		hr := F_VN_ResizeImage(ipImageIn,
							   ipImageForVideoRingBuffer,
							   ImageSmallWidth,
							   ImageSmallHeight,
							   1,
							   hr);
	ELSE
		hr := F_VN_CopyImage(ipImageIn, ipImageForVideoRingBuffer, hr);
	END_IF

	// Check to see if images are in memory
	//hr := FW_SafeRelease(ADR(BufferImageRing[BufferIndex]));
	//IF BufferImageRing[BufferIndex] <> 0 THEN
	//	FW_SafeRelease(ADR(BufferImageRing[BufferIndex]));
	//END_IF
	
	
	hrWD1		:= F_VN_StartRelWatchdog(tStop1, S_OK);
	hr			:= F_VN_CopyImage(ipImageForVideoRingBuffer, BufferImageRing[BufferIndex], S_OK);
	hrWD1		:= F_VN_StopWatchdog(hrWD1, tRest => tRest1);
	BufferIndex := BufferIndex + 1;
	IF BufferIndex > Parameters_Vision.MAX_NUMBER_IMAGES_2_VIDEO THEN
		BufferIndex := 1;
	END_IF
END_IF
END_METHOD

PROPERTY AlarmDelayTime : TIME
SET
_AlarmDelayTime := AlarmDelayTime;
END_SET
END_PROPERTY

PROPERTY CameraID : UINT
SET
_CameraID := CameraID;
END_SET
END_PROPERTY

PROPERTY FramesPerSecond : UINT
SET
_FramesPerSecond := FramesPerSecond;
END_SET
END_PROPERTY

PROPERTY ImageReductionFactor : LREAL
SET
_ImageReductionFactor := ImageReductionFactor;
END_SET
END_PROPERTY

PROPERTY ImageSourceDirectory : STRING
SET
_ImageSourceDirectory := ImageSourceDirectory;
END_SET
END_PROPERTY

PROPERTY VideoOutputDirectory : STRING
SET
_VideoOutputDirectory := VideoOutputDirectory;
END_SET
END_PROPERTY

METHOD WriteImage : BOOL
VAR_INPUT
	BufferImageSaveNameIndex : INT;
	Index					 : INT;
END_VAR

VAR
	SysTimeAtImageSave : ULINT;
END_VAR
CASE WriteFileState OF
	0:
		sImageToSaveName := CONCAT(STR1 := _ImageSourceDirectory, '\Image');
		CASE Index OF // Add leading zeros to index number of image name
			0..9:
				sImageToSaveName := CONCAT(sImageToSaveName, '000');
				sImageToSaveName := CONCAT(sImageToSaveName, ULINT_TO_STRING(Index));

			10..99:
				sImageToSaveName := CONCAT(sImageToSaveName, '00');
				sImageToSaveName := CONCAT(sImageToSaveName, ULINT_TO_STRING(Index));

			100..999:
				sImageToSaveName := CONCAT(sImageToSaveName, '0');
				sImageToSaveName := CONCAT(sImageToSaveName, ULINT_TO_STRING(Index));

		ELSE
			sImageToSaveName := CONCAT(sImageToSaveName, ULINT_TO_STRING(Index));
		END_CASE;

		sImageToSaveName	:= CONCAT(sImageToSaveName, '.png');
		ipImageToSave		:= BufferImageRing[BufferImageSaveNameIndex];
		SysTimeAtImageSave	:= F_GetSystemTime();
		WriteFileState		:= 10;

	10:
		// sFilePath must contain the full path, image name and type
		fbWriteImage(ipImage := ipImageToSave, sFilePath := sImageToSaveName, nTimeout := T#500MS,bWrite := TRUE);
		IF NOT fbWriteImage.bBusy THEN
			fbWriteImage(sFilePath := sImageToSaveName, bWrite := FALSE);
			WriteFileState := 0;
			WriteImage := TRUE;
		END_IF

ELSE
	WriteFileState := 0;
END_CASE

(*//bSaveImageNow := FALSE;
WriteImageWaitResult := TRUE;

// sFilePath must contain the full path, image name and type
fbWriteImage(ipImage   := ipImageToSave,
			 sFilePath := sImageToSaveName,
			 bWrite	   := TRUE,
			 nTimeout  := T#500MS);

IF NOT fbWriteImage.bBusy AND NOT fbWriteImage.bError THEN
	fbWriteImage(bWrite := FALSE, sFilePath := sImageToSaveName);
	WriteImage := TRUE;
END_IF*)
END_METHOD

END_FUNCTION_BLOCK

// Vision/VisionTask/FB_VisionCameraMonitor
FUNCTION_BLOCK FB_VisionCameraMonitor EXTENDS FB_VisionCameraBase
VAR
	// Video making properties
	_CameraID			  : UINT   := 1;
	_FramesPerSecond	  : UINT   := 10;
	_ImageSourceDirectory : STRING := 'C:\Images';
	_VideoOutputDirectory : STRING := 'C:\Videos';

	// Listener for JSON alarms with "Create
	VideoPlaybackControl :
		FB_VideoPlaybackControl := (ImageReductionFactor := 0.2, CameraID := _CameraID, ImageSourceDirectory := _ImageSourceDirectory,
									VideoOutputDirectory													 := _VideoOutputDirectory);
END_VAR

PROPERTY CameraID : UINT
SET
_CameraID := CameraID;
END_SET
END_PROPERTY

PROPERTY FramesPerSecond : UINT
SET
_FramesPerSecond := FramesPerSecond;
END_SET
END_PROPERTY

PROPERTY ImageSourceDirectory : STRING
SET
_ImageSourceDirectory := ImageSourceDirectory;
END_SET
END_PROPERTY

PROPERTY VideoOutputDirectory : STRING
SET
_VideoOutputDirectory := VideoOutputDirectory;
END_SET
END_PROPERTY

METHOD PUBLIC CyclicLogic
// Call the base here
SUPER^.CyclicLogic();

// Call the video playback here
VideoPlaybackControl.CyclicLogic();
END_METHOD

METHOD PROTECTED Initialize : BOOL
VAR_INPUT
END_VAR





Initialize := TRUE;
END_METHOD

METHOD PUBLIC  ProcessImage
hr := F_VN_GetPixelFormat(ipImageIn, PixelFormat, hr);
IF PixelFormat.nChannels = 3 THEN
	hr := F_VN_CopyImage(ipImageIn, ipImageRes, hr);
	hr := F_VN_ConvertColorSpace(ipImageRes,
								 ipImageIn,
								 TCVN_CST_RGB_TO_GRAY,
								 hr);
ELSE
	hr := F_VN_ConvertColorSpace(ipImageIn,
								 ipImageRes,
								 TCVN_CST_Gray_TO_RGB,
								 hr);
END_IF

// Display Input Image
hr := F_VN_CopyIntoDisplayableImage(ipImageIn, ipImageInDisp, hr);


VideoPlaybackControl.AddImage(ipImageIn := ipImageIn);
END_METHOD

END_FUNCTION_BLOCK
